Fanuc TP program (LS listing): calib_1.ls

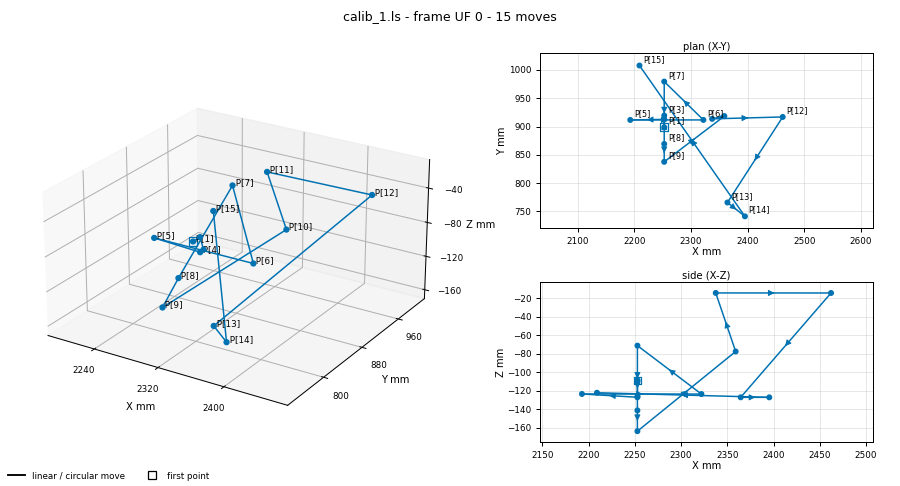
[picture p0: tool path of calib_1.ls in frame UF 0, 15 of 15 moves have a stored position in this frame; points joined in program order, loops and branches not executed]
/PROG  CALIB_1
/ATTR
OWNER		= MNEDITOR;
COMMENT		= "";
PROG_SIZE	= 1579;
CREATE		= DATE 25-09-25  TIME 19:15:44;
MODIFIED	= DATE 25-09-25  TIME 19:44:56;
FILE_NAME	= ;
VERSION		= 0;
LINE_COUNT	= 25;
MEMORY_SIZE	= 1851;
PROTECT		= READ_WRITE;
TCD:  STACK_SIZE	= 0,
      TASK_PRIORITY	= 50,
      TIME_SLICE	= 0,
      BUSY_LAMP_OFF	= 0,
      ABORT_REQUEST	= 0,
      PAUSE_REQUEST	= 0;
DEFAULT_GROUP	= 1,1,*,*,*;
CONTROL_CODE	= 00000000 00000000;
LOCAL_REGISTERS	= 0,0,0;
/MN
   1:  UFRAME_NUM=0 ;
   2:  UTOOL_NUM=10 ;
   3:  OVERRIDE=30% ;
   4:   ;
   5:L P[1] 100mm/sec FINE    ;
   6:L P[2] 100mm/sec FINE    ;
   7:L P[3] 100mm/sec FINE    ;
   8:   ;
   9:L P[4] 100mm/sec FINE    ;
  10:L P[5] 100mm/sec FINE    ;
  11:L P[6] 100mm/sec FINE    ;
  12:   ;
  13:L P[7] 100mm/sec FINE    ;
  14:L P[8] 100mm/sec FINE    ;
  15:L P[9] 100mm/sec FINE    ;
  16:   ;
  17:L P[10] 100mm/sec FINE    ;
  18:L P[11] 100mm/sec FINE    ;
  19:L P[12] 100mm/sec FINE    ;
  20:   ;
  21:L P[13] 100mm/sec FINE    ;
  22:L P[14] 100mm/sec FINE    ;
  23:L P[15] 100mm/sec FINE    ;
  24:   ;
  25:   ;
/POS
P[1]{
   GP1:
	UF : 0, UT : 10,		CONFIG : 'N U T, 0, 0, 0',
	X =  2252.764  mm,	Y =   898.654  mm,	Z =  -108.850  mm,
	W =  -179.972 deg,	P =     -.028 deg,	R =     -.549 deg
   GP2:
	UF : 0, UT : 10,
	J1=     -.082 deg
};
P[2]{
   GP1:
	UF : 0, UT : 10,		CONFIG : 'N U T, 0, 0, 0',
	X =  2252.733  mm,	Y =   912.646  mm,	Z =  -108.898  mm,
	W =  -179.973 deg,	P =     -.027 deg,	R =     -.548 deg
   GP2:
	UF : 0, UT : 10,
	J1=     -.082 deg
};
P[3]{
   GP1:
	UF : 0, UT : 10,		CONFIG : 'N U T, 0, 0, 0',
	X =  2252.748  mm,	Y =   919.452  mm,	Z =  -126.300  mm,
	W =  -179.973 deg,	P =     -.026 deg,	R =     -.549 deg
   GP2:
	UF : 0, UT : 10,
	J1=     -.082 deg
};
P[4]{
   GP1:
	UF : 0, UT : 10,		CONFIG : 'N U T, 0, 0, 0',
	X =  2252.709  mm,	Y =   912.691  mm,	Z =  -126.981  mm,
	W =  -179.973 deg,	P =     -.026 deg,	R =     -.547 deg
   GP2:
	UF : 0, UT : 10,
	J1=     -.082 deg
};
P[5]{
   GP1:
	UF : 0, UT : 10,		CONFIG : 'N U T, 0, 0, 0',
	X =  2192.736  mm,	Y =   911.611  mm,	Z =  -123.425  mm,
	W =  -179.974 deg,	P =     -.025 deg,	R =     -.548 deg
   GP2:
	UF : 0, UT : 10,
	J1=     -.082 deg
};
P[6]{
   GP1:
	UF : 0, UT : 10,		CONFIG : 'N U T, 0, 0, 0',
	X =  2321.923  mm,	Y =   911.661  mm,	Z =  -123.510  mm,
	W =  -179.974 deg,	P =     -.023 deg,	R =     -.547 deg
   GP2:
	UF : 0, UT : 10,
	J1=     -.082 deg
};
P[7]{
   GP1:
	UF : 0, UT : 10,		CONFIG : 'N U T, 0, 0, 0',
	X =  2252.732  mm,	Y =   979.445  mm,	Z =   -71.153  mm,
	W =   173.258 deg,	P =     -.088 deg,	R =     -.542 deg
   GP2:
	UF : 0, UT : 10,
	J1=     -.082 deg
};
P[8]{
   GP1:
	UF : 0, UT : 10,		CONFIG : 'N U T, 0, 0, 0',
	X =  2252.708  mm,	Y =   869.197  mm,	Z =  -141.203  mm,
	W =  -175.853 deg,	P =      .017 deg,	R =     -.548 deg
   GP2:
	UF : 0, UT : 10,
	J1=     -.082 deg
};
P[9]{
   GP1:
	UF : 0, UT : 10,		CONFIG : 'N U T, 0, 0, 0',
	X =  2252.684  mm,	Y =   837.642  mm,	Z =  -163.690  mm,
	W =  -171.941 deg,	P =      .055 deg,	R =     -.544 deg
   GP2:
	UF : 0, UT : 10,
	J1=     -.082 deg
};
P[10]{
   GP1:
	UF : 0, UT : 10,		CONFIG : 'N U T, 0, 0, 0',
	X =  2358.978  mm,	Y =   918.395  mm,	Z =   -77.469  mm,
	W =   179.971 deg,	P =     5.669 deg,	R =     -.549 deg
   GP2:
	UF : 0, UT : 10,
	J1=     -.082 deg
};
P[11]{
   GP1:
	UF : 0, UT : 10,		CONFIG : 'N U T, 0, 0, 0',
	X =  2337.435  mm,	Y =   913.531  mm,	Z =   -14.162  mm,
	W =   179.906 deg,	P =    12.149 deg,	R =     -.559 deg
   GP2:
	UF : 0, UT : 10,
	J1=     -.082 deg
};
P[12]{
   GP1:
	UF : 0, UT : 10,		CONFIG : 'N U T, 0, 0, 0',
	X =  2462.127  mm,	Y =   916.925  mm,	Z =   -14.211  mm,
	W =   179.878 deg,	P =    14.853 deg,	R =     -.567 deg
   GP2:
	UF : 0, UT : 10,
	J1=     -.082 deg
};
P[13]{
   GP1:
	UF : 0, UT : 10,		CONFIG : 'N U T, 0, 0, 0',
	X =  2364.417  mm,	Y =   765.753  mm,	Z =  -127.050  mm,
	W =  -179.974 deg,	P =     -.024 deg,	R =    17.723 deg
   GP2:
	UF : 0, UT : 10,
	J1=     -.082 deg
};
P[14]{
   GP1:
	UF : 0, UT : 10,		CONFIG : 'N U T, 0, 0, 0',
	X =  2395.335  mm,	Y =   741.284  mm,	Z =  -127.083  mm,
	W =  -179.974 deg,	P =     -.023 deg,	R =    21.411 deg
   GP2:
	UF : 0, UT : 10,
	J1=     -.082 deg
};
P[15]{
   GP1:
	UF : 0, UT : 10,		CONFIG : 'N U T, 0, 0, 0',
	X =  2208.990  mm,	Y =  1007.787  mm,	Z =  -122.089  mm,
	W =  -179.974 deg,	P =     -.024 deg,	R =   -10.906 deg
   GP2:
	UF : 0, UT : 10,
	J1=     -.082 deg
};
/END
